// TIA Portal V17 export
// export: Created 2025-03-07T09:24:31.5390516Z, ExportSetting WithDefaults, DisplayName Totally Integrated Automation Portal, DisplayVersion V17 Update 8, DisplayName TIA Portal Openness, DisplayVersion V17 Update 8, DisplayName TIA Portal Version Control Interface, DisplayVersion V17, DisplayName SINAMICS Startdrive Advanced, DisplayVersion V17 SP2, DisplayName SINAMICS Startdrive G110M, G120, G120C, G120D, G120P, G115D, DisplayVersion V17 SP2, DisplayName SINAMICS Startdrive G130, G150, S120, S150, SINAMICS MV, S210, DisplayVersion V17 SP2, DisplayName STEP 7 Professional, DisplayVersion V17 Update 8, DisplayName SINUMERIK ONE STEP 7 Toolbox, DisplayVersion V17 Update 12, DisplayName SINUMERIK 840D sl STEP 7 Toolbox, DisplayVersion V17 Update 12, DisplayName STEP 7 Safety, DisplayVersion V17 Update 6, DisplayName WinCC Advanced, DisplayVersion V17 Update 8
VAR_GLOBAL   // PLC tag table "TAGS_IO_GENERAL_CLADDING"
   "/////_CRM_/////" AT %M6060.0 : Bool;   // /////_CRM_/////
   "/////_ELECTRICAL_CABINET_/////" AT %M6100.0 : Bool;   // /////_ELECTRICAL_CABINET_/////
   "/////_LINE_CONTACTOR_/////" AT %M6200.0 : Bool;   // /////_LINE_CONTACTOR_/////
   "/////_MPP_AND_SIGNAL_TOWER_/////" AT %M141.0 : Bool;   // /////_MPP_AND_SIGNAL_TOWER_/////
   "/////_POWER_SUPPLY_/////" AT %M6080.0 : Bool;   // /////_POWER_SUPPLY_/////
   "/////_SAFETY_DOORS_/////" AT %M6180.0 : Bool;   // /////_SAFETY_DOORS_/////
   CIRCUIT_BREAKER_230VAC_TRIPPED AT %I140.1 : Bool;   // 230 VAC CIRCUIT BREAKER TRIPPED
   CIRCUIT_BREAKER_FC04_TRIPPED AT %I140.0 : Bool;   // FC04 CIRCUIT BREAKER TRIPPED. FAN.
   CIRCUIT_BREAKER_FC35_1_TRIPPED AT %I140.5 : Bool;   // FC35.1 CIRCUIT BREAKER TRIPPED
   CIRCUIT_BREAKER_FC35_2_TRIPPED AT %I140.6 : Bool;   // FC35.2 CIRCUIT BREAKER TRIPPED
   CIRCUIT_BREAKER_FC35_3_TRIPPED AT %I140.7 : Bool;   // FC35.3 CIRCUIT BREAKER TRIPPED
   CONTROL_ON_Q AT %Q140.0 : Bool;   // CONTROL ON OUTPUT
   MAIN_CIRCUIT_BREAKER_I AT %M580.1 : Bool;   // MAIN CABINET CIRCUIT BREAKER TRIPPED INPUT
   PB_AUTO_CYCLE_LIGHT_Q AT %Q141.1 : Bool;   // AUTOMATIC CYCLE LIGHT OUTPUT
   PB_AUTO_MODE_SELECTED_LIGHT_Q AT %Q141.2 : Bool;   // AUTOMATIC MODE SELECTED LIGHT OUTPUT
   PB_IMMEDIATE_STOP_I AT %I144.3 : Bool;   // IMMEDIATE STOP INPUT
   PB_MANUAL_MODE_SELECTED_LIGHT_Q AT %Q141.3 : Bool;   // MANUAL MODE SELECTED LIGHT OUTPUT
   PB_RESET_FAULTS_I AT %I144.6 : Bool;   // RESET FAULTS INPUT
   PB_START_CYCLE_I AT %I144.2 : Bool;   // START CYCLE INPUT
   PS_24V_NOT_READY_DEV_1_I AT %I142.2 : Bool;   // POWER SUPPLY 24V NOT READY DEVICE 1 INPUT
   PS_24V_NOT_READY_DEV_2_I AT %I142.3 : Bool;   // POWER SUPPLY 24V NOT READY DEVICE 2 INPUT
   SIGNAL_TWR_BLUE_LIGHT_Q AT %M141.1 : Bool;   // SIGNAL TOWER BLUE LIGHT OUTPUT
   SIGNAL_TWR_GREEN_LIGHT_Q AT %Q141.5 : Bool;   // SIGNAL TOWER GREEN LIGHT OUTPUT
   SIGNAL_TWR_HOOTER_Q AT %M141.3 : Bool;   // SIGNAL TOWER HOOTER LIGHT OUTPUT
   SIGNAL_TWR_RED_LIGHT_Q AT %Q141.7 : Bool;   // SIGNAL TOWER RED LIGHT OUTPUT
   SIGNAL_TWR_WHITE_LIGHT_Q AT %M141.2 : Bool;   // SIGNAL TOWER WHITE LIGHT OUTPUT
   SIGNAL_TWR_YELLOW_LIGHT_Q AT %Q141.6 : Bool;   // SIGNAL TOWER YELLOW LIGHT OUTPUT
   PB_HOPPERS_AUTO_MODE_SELECTED_LIGHT_Q AT %Q141.0 : Bool;   // AUTOMATIC MODE SELECTED LIGHT OUTPUT
   PB_FEEDERS_AUTOMATIC_MODE_SELECT_I AT %I144.0 : Bool;   // AUTOMATIC MODE SELECT INPUT
   PB_FEEDERS_MANUAL_MODE_SELECT_I AT %I144.1 : Bool;   // MANUAL MODE SELECT INPUT
   PB_HOPPERS_MANUAL_MODE_SELECT_I AT %I142.6 : Bool;   // MANUAL MODE SELECT INPUT
   PB_HOPPERS_AUTOMATIC_MODE_SELECT_I AT %I142.5 : Bool;   // AUTOMATIC MODE SELECT INPUT
END_VAR
